Staubli VAL3: isDetected.pgx

public program isDetected(num& x_nHowMany[] (dimensions=1))
begin
  x_nHowMany=nNumOfPart
end
